FUNCTION_BLOCK EA_network2
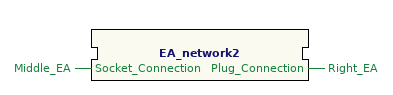
  SOCKETS
    Socket_Connection : Middle_EA;
  END_SOCKETS
  PLUGS
    Plug_Connection : Right_EA;
  END_PLUGS
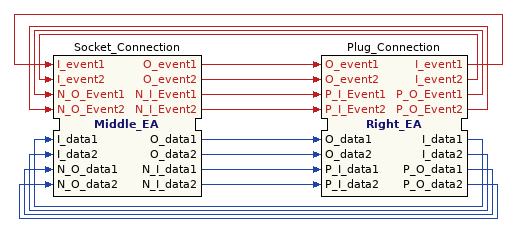
  EVENT_CONNECTIONS
    Socket_Connection.O_event1 TO Plug_Connection.O_event1;
    Socket_Connection.O_event2 TO Plug_Connection.O_event2;
    Socket_Connection.N_I_Event1 TO Plug_Connection.P_I_Event1;
    Socket_Connection.N_I_Event2 TO Plug_Connection.P_I_Event2;
    Plug_Connection.I_event1 TO Socket_Connection.I_event1;
    Plug_Connection.I_event2 TO Socket_Connection.I_event2;
    Plug_Connection.P_O_Event1 TO Socket_Connection.N_O_Event1;
    Plug_Connection.P_O_Event2 TO Socket_Connection.N_O_Event2;
  END_CONNECTIONS
  DATA_CONNECTIONS
    Socket_Connection.O_data1 TO Plug_Connection.O_data1;
    Socket_Connection.O_data2 TO Plug_Connection.O_data2;
    Socket_Connection.N_I_data1 TO Plug_Connection.P_I_data1;
    Socket_Connection.N_I_data2 TO Plug_Connection.P_I_data2;
    Plug_Connection.I_data1 TO Socket_Connection.I_data1;
    Plug_Connection.I_data2 TO Socket_Connection.I_data2;
    Plug_Connection.P_O_data1 TO Socket_Connection.N_O_data1;
    Plug_Connection.P_O_data2 TO Socket_Connection.N_O_data2;
  END_CONNECTIONS
END_FUNCTION_BLOCK
